{attribute 'qualified_only'}
VAR_GLOBAL
		EtherCAT_Master_AMIxxxx : EtherCAT_Master_AMIxxxx_CEFF3AAB;
END_VAR

(* stored: Version 1.2.0.0, ProductVersion 3.1.4024.9
   GVL GVL_iXlinker: Id {d93a9623-0f49-4b45-90d8-b241f5225215} *)
